// TIA Portal V21 export
FUNCTION "GestMotore_GestQuota" : Void   // FC40, LAD
{ S7_Optimized_Access := 'TRUE' }
// stored: SetENOAutomatically false
   VAR_INPUT
      K_Quota : Int;
      K_Motore : Int;
      CondizioniQuota : Bool;
      Quota : Real;
   END_VAR
   VAR_TEMP
      FinestraInPosizione_Pos : Real;
      FinestraInPosizione_Neg : Real;
      PosAttualeMotore : Real;
   END_VAR
BEGIN

REGION Network 1: Passo al motore la quota richiesta
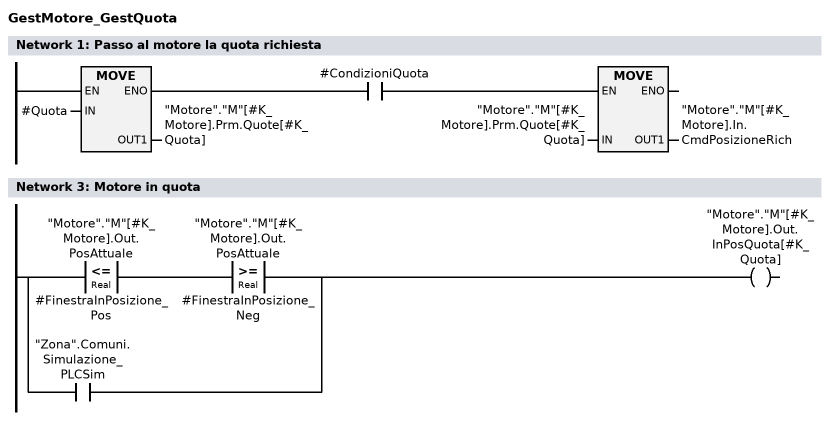
   RUNG wire#powerrail
      Move(in := #Quota, out1 => "Motore"."M"[#K_Motore].Prm.Quote[#K_Quota])
      Contact( #CondizioniQuota )
      Move(in := "Motore"."M"[#K_Motore].Prm.Quote[#K_Quota], out1 => "Motore"."M"[#K_Motore].In.CmdPosizioneRich)
   END_RUNG
   // the same network as SCL:
   "Motore"."M"[#K_Motore].Prm.Quote[#K_Quota] := #Quota;
   IF #CondizioniQuota THEN
       "Motore"."M"[#K_Motore].In.CmdPosizioneRich := "Motore"."M"[#K_Motore].Prm.Quote[#K_Quota];
   END_IF;
END_REGION

REGION Network 2 (SCL): Calcolo quote finestra
   #FinestraInPosizione_Pos := "Motore".M[#K_Motore].Prm.Quote[#K_Quota] + "Motore".M[#K_Motore].Prm.Posizionatore.DeadBand_InPosition;
   #FinestraInPosizione_Neg := "Motore".M[#K_Motore].Prm.Quote[#K_Quota] - "Motore".M[#K_Motore].Prm.Posizionatore.DeadBand_InPosition;
END_REGION

REGION Network 3: Motore in quota
   RUNG wire#powerrail
      { S7_Templates := "SrcType := Real" } LE_Contact(in1 := "Motore"."M"[#K_Motore].Out.PosAttuale, in2 := #FinestraInPosizione_Pos)
      { S7_Templates := "SrcType := Real" } GE_Contact(in1 := "Motore"."M"[#K_Motore].Out.PosAttuale, in2 := #FinestraInPosizione_Neg)
      wire#w1
      Coil( "Motore"."M"[#K_Motore].Out.InPosQuota[#K_Quota] )
   END_RUNG
   RUNG wire#powerrail
      Contact( "Zona".Comuni.Simulazione_PLCSim )
   END_RUNG wire#w1
   // the same network as SCL:
   "Motore"."M"[#K_Motore].Out.InPosQuota[#K_Quota] := (("Motore"."M"[#K_Motore].Out.PosAttuale <= #FinestraInPosizione_Pos) AND ("Motore"."M"[#K_Motore].Out.PosAttuale >= #FinestraInPosizione_Neg)) OR "Zona".Comuni.Simulazione_PLCSim;
END_REGION
END_FUNCTION
